(* CODESYS project sensata_lasermarker.library
   Company: Sensata Technologies
   DocFormat: reStructuredText
   Description: This library is for the Laser Markers.
   Version: 0.0.1
   Placeholder: Sensata_LaserMarker
   Title: Sensata_LaserMarker

Project tree, tasks and I/O mapping:
  libraries: Sensata_Common, * (Sensata Technologies); Sensata_Utilities, * (Sensata Technologies); Tc2_Standard, * (Beckhoff Automation GmbH); Tc2_System, * (Beckhoff Automation GmbH); Tc2_Utilities, * (Beckhoff Automation GmbH); Tc3_Module, * (Beckhoff Automation GmbH); Sensata_Vision, * (Sensata Technologies)
  Abstract/
    function block FB_LaserMarker [ST]
  Concrete/
    function block FB_KeyenceLaserMarkerMDX2000 [LD]: M_Connect, M_Disconnect, M_GetConnectStatus, P_bConnectBusy, P_bConnected, M_PeakCurrentProgram, M_GetCurrentProgram, M_GetProgramState, M_LoadProgram, M_PauseProgram, M_SaveCurrentLaserProgramtoPC, M_SendProgramtoLaser, M_StartMarking, M_StartProgram, M_StopMarking, M_StopProgram, M_UpdateProgramBlockInTheLaser, P_bProgramControlBusy, P_enumProgramState, P_strCurrentProgram, M_GetAllLaserErrorStatus, M_GetAllLaserStatus, M_ClearLaserErrors, M_Reset, P_bResetBusy, M_Trigger, P_bTriggerBusy, M_HandleCommand
  Interfaces/
    interface I_Markable: StartMarking, StopMarking
  Project Information/
    function F_GetCompany [ST]
    function F_GetTitle [ST]
    function F_GetVersion [ST]
  Version/
    global variables Global_Version
  global variables GVL_LaserMarker
*)

// Version/Global_Version
{attribute 'TcGenerated'}
{attribute 'no-analysis'}
{attribute 'linkalways'}
// This function has been automatically generated from the project information.
VAR_GLOBAL CONSTANT
	{attribute 'const_non_replaced'}
	stLibVersion_Sensata_LaserMarker : ST_LibVersion := (iMajor := 0, iMinor := 0, iBuild := 1, iRevision := 0, nFlags := 0, sVersion := '0.0.1');
END_VAR

// GVL_LaserMarker
VAR_GLOBAL
	LaserConnected : BOOL := FALSE;
	PeakCurrentProgramSuccess : BOOL := FALSE;
	SendProgramToLaserSuccess : BOOL := FALSE;
END_VAR

// Abstract/FB_LaserMarker
FUNCTION_BLOCK ABSTRACT FB_LaserMarker EXTENDS FB_Device
VAR_INPUT
END_VAR
VAR_OUTPUT
END_VAR
VAR
END_VAR

END_FUNCTION_BLOCK

// Concrete/FB_KeyenceLaserMarkerMDX2000
FUNCTION_BLOCK PUBLIC FB_KeyenceLaserMarkerMDX2000 EXTENDS FB_LaserMarker
	IMPLEMENTS 
		I_Connectable,
		I_Resettable,
		I_Programmable,
		I_Triggerable
VAR_INPUT
	fbApi : REFERENCE TO FB_AdsCommandRouter; (* Device API connection to the "". *)
END_VAR
VAR_OUTPUT
END_VAR
VAR
	// Connectable
	bApiConnected: BOOL; (* TRUE if the API is connected. *)
	bConnected: BOOL; (* TRUE if the Laser is connected. *)
	bConnecting: BOOL; (* TRUE while the connect command is running. *)
	bDisconnecting: BOOL; (* TRUE while the disconnect command is running. *)
	bActive: BOOL;
   bSendingSendLaserProgram : BOOL;
	
	//Laser Related Variables
	
	ADSRouter: Sensata_Utilities.FB_AdsCommandRouter;
END_VAR

// NETWORK 1

METHOD M_Connect : BOOL
VAR_INPUT
	
END_VAR
VAR_OUTPUT
	
END_VAR
VAR
	bApiResult: BOOL;
	arrParameters: T_ApiMethodParameters;
	bContinue: BOOL;
	bCommandResult: BOOL;
	bCommandSent: BOOL;
	strReturn: STRING(255);
	bMethodCalled: BOOL;
	udintErrorCode: UDINT;
	strErrorMessage: T_MaxString;
	strResult : T_MaxString;

    buildArray: BOOL;    
    doIt: BOOL;
    buildArrayDB: BOOL;
    tagName: STRING := 'strProc';
    sataType: STRING := 'String';
    arrParams: T_ApiParameterList;
    
    doReset: BOOL;
    
    strTarget: T_MaxString := 'Laser_1';//'PAC_1';
    strCommand: T_MaxString := 'Connect';//'Write';
//    strProc: T_MaxString := 'spInsert';
    
    paramDictionary : T_ApiParameterList;
    p1: T_MaxString := 'MyMachine';
    p2: T_MaxString := 'MyLocation';
    p3: T_MaxString := 'MyPC';



   strRet: T_MaxString;
    adsRouter: FB_AdsCommandRouter;
    bResult: BOOL;
    arrOutputs: T_ApiParameterList;
    bExecuted: BOOL;
    
    pBuilder: FB_ApiParamBuilder;
    pArray: Sensata_Utilities.UXINT;
//    stTest: ST_TestStruct;



END_VAR
//M_Connect := FALSE;
//IF NOT bApiConnected THEN
//	bApiConnected := fbApi.M_Connect();
//END_IF
//udintErrorCode := 100;
//strErrorMessage := 'Error While connecting to Laser Marker';

//IF bApiConnected THEN
//	IF NOT fbApi.P_bDeviceInterfaceBusy OR bActive THEN
//		// Set continue to true
//		bActive := TRUE;
		
//		// Send command to API
////		bApiResult := fbApi.M_CallMethod(THIS^.in_strUniqueId, 'ConnectToLaserMarker' , arrParameters, strReturn => strResult);
//		bApiResult := fbApi.M_CallMethod(THIS^.in_strUniqueId, 'Connect' , arrParameters, strReturn => strResult);
		
//		IF NOT fbApi.P_bDeviceInterfaceBusy THEN
//			// Set continue to false
//			bActive := FALSE;
			
//			// Throw an error if the API has an error
//			IF fbApi.P_bError THEN
//				THIS^.M_SetError(
//					udintErrorCode,
//					strErrorMessage);
//			// If result is successful, set results accordingly
//			ELSIF bApiResult AND GVL_LaserMarker.LaserConnected THEN
//				M_Connect := TRUE;
//			END_IF
//		END_IF
//	END_IF
//END_IF


//Copied from Sensata_Test (Aiswarya)
//IF NOT bApiConnected THEN
//	bApiConnected := fbApi.M_Connect();
//END_IF

//bCommandResult := THIS^.M_HandleCommand(
//	THIS^.in_strUniqueId,
//	'Connect',
//	arrParameters,
//	//E_VitrekV70_Error.Connect,
//	100,
//	'Error while trying to connect to laser!',
//	bConnecting,
//	bContinue => bContinue);

//M_Connect := FALSE;
//IF bContinue THEN
//	bConnecting := TRUE;
//ELSIF bCommandResult THEN
//	bConnected := TRUE;
//	M_Connect := TRUE;
//END_IF


//Kevin's new ADS Server logic


IF doReset THEN
    doReset := FALSE;
    doIt := FALSE;
    adsRouter.M_ClearError();
END_IF

IF buildArray THEN
    pBuilder.M_ClearParameters();
//    pBuilder.M_AddParameter('tName', tagName);
//    pBuilder.M_AddParameter('dType', sataType);
    //pBuilder.M_AddParameter('retObj', NULL);
    pBuilder.M_OutputToParameterList(arrParams);
    buildArray := FALSE;
END_IF

//IF buildArrayDB THEN
//    pBuilder.M_ClearParameters();
//    pBuilder.M_AddParameter('procName', strProc);
//    pArray := pBuilder.M_AddParameter('paramDictionary', stTest);
//    pBuilder.M_AddStructMember(pArray,'@MachineName',p1);
//    pBuilder.M_AddStructMember(pArray,'@Location',p2);
//    pBuilder.M_AddStructMember(pArray,'@PCName',p3);
//    pBuilder.M_OutputToParameterList(arrParams);
//    buildArrayDB := FALSE;
//END_IF

//strTarget is 'Laser_1' in this case
//strCommand is 'Connect' in this case
//arrParams needs to be built using array builder


IF doIt THEN
    bResult := adsRouter.M_RouteCommand
      (
        strTarget, 
        strCommand, 
        T#5S, 
        arrParams, 
        arrOutputs, 
        _out_bCommandExecuted => bExecuted, 
        _out_strReturnValue => strRet
      );
    IF bExecuted THEN
        doIt := FALSE;
    END_IF  
END_IF
END_METHOD

METHOD PUBLIC M_Disconnect : BOOL
VAR
	arrParameters : T_ApiMethodParameters;
	bCommandResult : BOOL;
	bContinue : BOOL;
	bApiResult: BOOL;
	udintErrorCode: UDINT;
	strReturn: STRING(255);
	strResult : T_MaxString;
	strErrorMessage: T_MaxString;
END_VAR
//M_Disconnect := FALSE;
//IF NOT bApiConnected THEN
//	bApiConnected := fbApi.M_Connect();
//END_IF

//udintErrorCode := 101;
//strErrorMessage := 'Error While Disconnecting from Laser Marker';

//IF bApiConnected THEN
//	IF NOT fbApi.P_bDeviceInterfaceBusy OR bActive THEN
//		// Set continue to true
//		bActive := TRUE;
		
//		// Send command to API
//		//bApiResult := fbApi.M_CallMethod(THIS^.in_strUniqueId, 'DisconnectFromLaserMarker' , arrParameters, strReturn => strResult);
//		bApiResult := fbApi.M_CallMethod(THIS^.in_strUniqueId, 'Disconnect' , arrParameters, strReturn => strResult);
		
//		IF NOT fbApi.P_bDeviceInterfaceBusy THEN
//			// Set continue to false
//			bActive := FALSE;
//			// Throw an error if the API has an error
//			IF fbApi.P_bError THEN
//				THIS^.M_SetError( udintErrorCode, strErrorMessage);
//			ELSIF bApiResult THEN // If result is successful, set results accordingly
//				M_Disconnect := TRUE;
//			END_IF
//		END_IF
//	END_IF
//END_IF
END_METHOD

{warning 'add method implementation '}
(* This method should explicitly check the connection status of the device.
	Once the connection status is known, this method should return TRUE.
	If this method fails, P_bConnected should be set to FALSE since the device
	is not absolutely known to still be connected. *)
METHOD M_GetConnectStatus : BOOL
VAR_OUTPUT
	(* This should return TRUE if all connections required to make the device
		function properly are known to be connected, and FALSE otherwise. *)
	bConnected	: BOOL;
END_VAR
bConnected := P_bConnected;
M_GetConnectStatus := TRUE;
THIS^.M_LogWarning('Get connect status not implemented in UR e-Series!');
END_METHOD

(* This property should be TRUE while any method in this interface is actively
	executing, or FALSE otherwise. *)
PROPERTY P_bConnectBusy : BOOL
GET
P_bConnectBusy := bConnecting OR bDisconnecting;
END_GET
END_PROPERTY

(* This should be set to TRUE if M_Connect is successful or M_GetConnectStatus
	determines the device to be connected, and set to FALSE if M_Disconnect is
	called at all, M_GetConnectStatus fails, or M_GetConnectStatus determines
	the device to be not connected. *)
PROPERTY P_bConnected : BOOL
GET
P_bConnected := bApiConnected AND bConnected;
END_GET
END_PROPERTY

METHOD PUBLIC M_PeakCurrentProgram : BOOL
VAR_INPUT
END_VAR
VAR
	arrParameters : T_ApiMethodParameters;
	bApiResult: BOOL;
	udintErrorCode: UDINT;
	strErrorMessage: T_MaxString;
	strResult: T_MaxString;
END_VAR
//M_PeakCurrentProgram := FALSE;
//IF NOT bApiConnected THEN
//	bApiConnected := fbApi.M_Connect();
//END_IF

//udintErrorCode := 300;
//strErrorMessage := 'Error While performing M_PeakCurrentProgram function with Laser Marker';

//IF bApiConnected THEN
//	IF NOT fbApi.P_bDeviceInterfaceBusy OR bActive THEN
//		// Set continue to true
//		bActive := TRUE;
//		// Send command to API
//		bApiResult := fbApi.M_CallMethod(THIS^.in_strUniqueId, 'PeakCurrentProgram' , arrParameters, strReturn => strResult);
		
//		IF NOT fbApi.P_bDeviceInterfaceBusy THEN
//			// Set continue to false
//			bActive := FALSE;
//			// Throw an error if the API has an error
//			IF fbApi.P_bError THEN
//				THIS^.M_SetError( udintErrorCode, strErrorMessage);
//			ELSIF bApiResult THEN // If result is successful, set results accordingly
//				M_PeakCurrentProgram := TRUE;
//			END_IF
//		END_IF
//	END_IF
//END_IF
END_METHOD

{warning 'add method implementation '}
(* This method should explicitly get the current program loaded on the device.
	If the current program is successfully gotten, this method should return
	TRUE and set P_strCurrentProgram and strCurrentProgram to the gotten
	program name. If this method fails, both should be set to empty strings. *)
METHOD M_GetCurrentProgram : BOOL
VAR_OUTPUT
	(* This should be set to the name of the currently loaded program if
		the method was successful, or a blank string otherwise. *)
	strCurrentProgram	: Sensata_Common.T_MaxString;
END_VAR
END_METHOD

{warning 'add method implementation '}
(* This method should explicitly check the program state of the device.
	Once the program state is known, this method should return TRUE and set
	P_enumProgramState and enumProgramState to the relevant E_ProgramState
	value, else it should set both to E_ProgramState.Unknown. *)
METHOD M_GetProgramState : BOOL
VAR_OUTPUT
	(* If the program state is successfully gotten, this should be set to
		the relevant E_ProgramState value. If this method fails, this should
		be set to E_ProgramState.Unknown. *)
	enumProgramState	: Sensata_Common.E_ProgramState;
END_VAR
END_METHOD

{warning 'add method implementation '}
(* This method should load a new program onto the device, and then return TRUE
	once program loading is completed. Once this method begins the program loading
	process, P_strCurrentProgram should be cleared unless it is still explicitly
	known to be loaded. *)
METHOD M_LoadProgram : BOOL
VAR_INPUT
	(* String representing the program to load. If string must be in a specific
		format, make sure to override this comment to document it. *)
	strProgram	: Sensata_Common.T_MaxString;
END_VAR
END_METHOD

{warning 'add method implementation '}
(* This program should move to the program state from whatever state it was in
	to the Paused state, and then return TRUE once successful. If the program
	state is Stopped, this method should return TRUE but keep the current state
	as Stopped, since Paused at the beginning at the program is equivalent to
	being Stopped. *)
METHOD M_PauseProgram : BOOL
END_METHOD

METHOD PUBLIC M_SaveCurrentLaserProgramtoPC : BOOL
VAR_INPUT
	LaserProgramFolderPath : STRING;
END_VAR
VAR
	arrParameters : T_ApiMethodParameters;
	bApiResult: BOOL;
	udintErrorCode: UDINT;
	strErrorMessage: T_MaxString;
	strResult: T_MaxString;
END_VAR
//M_SaveCurrentLaserProgramtoPC := FALSE;
//IF NOT bApiConnected THEN
//	bApiConnected := fbApi.M_Connect();
//END_IF

//udintErrorCode := 200;
//strErrorMessage := 'Error While performing M_SaveCurrentLaserProgramtoPC from Laser Marker';

//IF bApiConnected THEN
//	IF NOT fbApi.P_bDeviceInterfaceBusy OR bActive THEN
//		// Set continue to true
//		bActive := TRUE;
//		arrParameters[1][1] := 'LaserProgramFolderPath';
//		arrParameters[1][2] := LaserProgramFolderPath;
//		// Send command to API
//		bApiResult := fbApi.M_CallMethod(THIS^.in_strUniqueId, 'SendProgramtoLaser' , arrParameters, strReturn => strResult);
		
//		IF NOT fbApi.P_bDeviceInterfaceBusy THEN
//			// Set continue to false
//			bActive := FALSE;
//			// Throw an error if the API has an error
//			IF fbApi.P_bError THEN
//				THIS^.M_SetError( udintErrorCode, strErrorMessage);
//			ELSIF bApiResult THEN // If result is successful, set results accordingly
//				M_SaveCurrentLaserProgramtoPC := TRUE;
//			END_IF
//		END_IF
//	END_IF
//END_IF
END_METHOD

METHOD PUBLIC M_SendProgramtoLaser : BOOL
VAR_INPUT
	filepath : STRING;
	LaserMemoryLocation : INT;
END_VAR
VAR
	bApiResult: BOOL;
	arrParameters: T_ApiMethodParameters;
	strResult: T_MaxString;
	udintErrorCode: UDINT;
	strErrorMessage: T_MaxString;
	bCommandResult : BOOL;
    bContinue: BOOL;
END_VAR
////M_SendProgramtoLaser := FALSE;
////IF NOT bApiConnected THEN
////	bApiConnected := fbApi.M_Connect();
////END_IF

//udintErrorCode := 201;
//strErrorMessage := 'Error While performing M_SendProgramtoLaser from Laser Marker';

////IF bApiConnected THEN
////	IF NOT fbApi.P_bDeviceInterfaceBusy OR bActive THEN
////		// Set continue to true
////		bActive := TRUE;
////		arrParameters[1][1] := 'filepath';
////		arrParameters[1][2] := filepath;
////		arrParameters[2][1] := 'LaserMemoryLocation';
////		arrParameters[2][2] := TO_STRING(LaserMemoryLocation);
////		// Send command to API
////		bApiResult := fbApi.M_CallMethod(THIS^.in_strUniqueId, 'SendProgramtoLaser' , arrParameters, strReturn => strResult);
		
////		IF NOT fbApi.P_bDeviceInterfaceBusy THEN
////			// Set continue to false
////			bActive := FALSE;
////			// Throw an error if the API has an error
////			IF fbApi.P_bError THEN
////				THIS^.M_SetError( udintErrorCode, strErrorMessage);
////			ELSIF bApiResult AND GVL_LaserMarker.SendProgramToLaserSuccess THEN // If result is successful, set results accordingly
////				M_SendProgramtoLaser := TRUE;
////			END_IF
////		END_IF
////	END_IF
////END_IF


////Copied from Aish

//		arrParameters[1][1] := 'filepath';
//		arrParameters[1][2] := filepath;
//		arrParameters[2][1] := 'LaserMemoryLocation';
//		arrParameters[2][2] := TO_STRING(LaserMemoryLocation);

//bCommandResult := THIS^.M_HandleCommand(
//    THIS^.in_strUniqueId,
//    'SendProgramtoLaser',
//    arrParameters,
//    udintErrorCode,
//    strErrorMessage,
//    bSendingSendLaserProgram,
//    bContinue => bContinue);
//M_SendProgramtoLaser := FALSE;
//IF bContinue THEN
//    bSendingSendLaserProgram := TRUE;
//ELSIF bCommandResult THEN
//        M_SendProgramtoLaser := TRUE;
//END_IF
END_METHOD

METHOD PUBLIC M_StartMarking : BOOL
VAR_INPUT
END_VAR

VAR
	bApiResult: BOOL;
	arrParameters: T_ApiMethodParameters;
	strResult: T_MaxString;
	udintErrorCode: UDINT;
	strErrorMessage: T_MaxString;
END_VAR
//M_StartMarking := FALSE;
//IF NOT bApiConnected THEN
//	bApiConnected := fbApi.M_Connect();
//END_IF

//udintErrorCode := 202;
//strErrorMessage := 'Error While performing M_StartMarking from Laser Marker';

//IF bApiConnected THEN
//	IF NOT fbApi.P_bDeviceInterfaceBusy OR bActive THEN
//		// Set continue to true
//		bActive := TRUE;
//		// Send command to API
//		bApiResult := fbApi.M_CallMethod(THIS^.in_strUniqueId, 'StartMarking' , arrParameters, strReturn => strResult);
		
//		IF NOT fbApi.P_bDeviceInterfaceBusy THEN
//			// Set continue to false
//			bActive := FALSE;
//			// Throw an error if the API has an error
//			IF fbApi.P_bError THEN
//				THIS^.M_SetError( udintErrorCode, strErrorMessage);
//			ELSIF bApiResult THEN // If result is successful, set results accordingly
//				M_StartMarking := TRUE;
//			END_IF
//		END_IF
//	END_IF
//END_IF
END_METHOD

{warning 'add method implementation '}
(* This should move the program state from whatever state it is in to the
	Running state, and then return TRUE once successful. Starting from the
	Paused state should always continue execution from whatever point the
	program was at when the program was initially paused. *)
METHOD M_StartProgram : BOOL
END_METHOD

METHOD PUBLIC M_StopMarking : BOOL
VAR_INPUT
END_VAR
VAR
	bApiResult: BOOL;
	arrParameters: T_ApiMethodParameters;
	strResult: T_MaxString;
	udintErrorCode: UDINT;
	strErrorMessage: T_MaxString;
END_VAR
//M_StopMarking := FALSE;
//IF NOT bApiConnected THEN
//	bApiConnected := fbApi.M_Connect();
//END_IF

//udintErrorCode := 203;
//strErrorMessage := 'Error While performing M_StopMarking from Laser Marker';

//IF bApiConnected THEN
//	IF NOT fbApi.P_bDeviceInterfaceBusy OR bActive THEN
//		// Set continue to true
//		bActive := TRUE;
//		// Send command to API
//		bApiResult := fbApi.M_CallMethod(THIS^.in_strUniqueId, 'StopMarking' , arrParameters, strReturn => strResult);
		
//		IF NOT fbApi.P_bDeviceInterfaceBusy THEN
//			// Set continue to false
//			bActive := FALSE;
//			// Throw an error if the API has an error
//			IF fbApi.P_bError THEN
//				THIS^.M_SetError( udintErrorCode, strErrorMessage);
//			ELSIF bApiResult THEN // If result is successful, set results accordingly
//				M_StopMarking := TRUE;
//			END_IF
//		END_IF
//	END_IF
//END_IF
END_METHOD

{warning 'add method implementation '}
(* This should change the program state from whatever state it was in to the
	Stopped state and then return TRUE. Moving to the Stopped state should
	always reset the program execution back to the beginning. *)
METHOD M_StopProgram : BOOL
END_METHOD

METHOD PUBLIC M_UpdateProgramBlockInTheLaser : BOOL
VAR_INPUT
	LaserProgramMemoryLocation : INT;
	BlockNumber : INT;
	BlockData : STRING;
	BlockType : BlockTypes;
END_VAR
VAR
	bApiResult: BOOL;
	arrParameters: T_ApiMethodParameters;
	strResult: T_MaxString;
	udintErrorCode: UDINT;
	strErrorMessage: T_MaxString;
END_VAR
//M_UpdateProgramBlockInTheLaser := FALSE;
//IF NOT bApiConnected THEN
//	bApiConnected := fbApi.M_Connect();
//END_IF

//udintErrorCode := 204;
//strErrorMessage := 'Error While performing M_UpdateProgramBlockInTheLaser from Laser Marker';

//IF bApiConnected THEN
//	IF NOT fbApi.P_bDeviceInterfaceBusy OR bActive THEN
//		// Set continue to true
//		bActive := TRUE;
//		arrParameters[1][1] := 'LaserProgramMemoryLocation';
//		arrParameters[1][2] := TO_STRING(LaserProgramMemoryLocation);
//		arrParameters[2][1] := 'BlockNumber';
//		arrParameters[2][2] := TO_STRING(BlockNumber);
//		arrParameters[3][1] := 'BlockData';
//		arrParameters[3][2] := BlockData;
//		arrParameters[4][1] := 'BlockType';
//		arrParameters[4][2] := TO_STRING(BlockType);
		
//		// Send command to API
//		bApiResult := fbApi.M_CallMethod(THIS^.in_strUniqueId, 'UpdateSingleBlockInTheLaserProgram' , arrParameters, strReturn => strResult);
		
//		IF NOT fbApi.P_bDeviceInterfaceBusy THEN
//			// Set continue to false
//			bActive := FALSE;
//			// Throw an error if the API has an error
//			IF fbApi.P_bError THEN
//				THIS^.M_SetError( udintErrorCode, strErrorMessage);
//			ELSIF bApiResult THEN // If result is successful, set results accordingly
//				M_UpdateProgramBlockInTheLaser := TRUE;
//			END_IF
//		END_IF
//	END_IF
//END_IF
END_METHOD

(* This property should be TRUE while any method in this interface is actively
	executing, or FALSE otherwise. *)
PROPERTY P_bProgramControlBusy : BOOL
GET
END_GET
END_PROPERTY

(* The current E_ProgramState value of the device. This should be reset to
	E_ProgramState.Unknown if any methods in this interface interact with the
	device but fail. *)
PROPERTY P_enumProgramState : Sensata_Common.E_ProgramState
GET
END_GET
END_PROPERTY

(* The value of the currently loaded program. This should only be set by
	M_LoadProgram or M_GetCurrentProgram, and set to a blank string if either
	fail. *)
PROPERTY P_strCurrentProgram : Sensata_Common.T_MaxString
GET
END_GET
END_PROPERTY

METHOD PUBLIC M_GetAllLaserErrorStatus : BOOL
VAR_INPUT
END_VAR
END_METHOD

METHOD PUBLIC M_GetAllLaserStatus : BOOL
VAR_INPUT
END_VAR
END_METHOD

METHOD PUBLIC M_ClearLaserErrors : BOOL
VAR
	arrParameters : T_ApiMethodParameters;
	bApiResult: BOOL;
	udintErrorCode: UDINT;
//	strReturn: STRING(255);
	strResult : T_MaxString;
	strErrorMessage: T_MaxString;
END_VAR
//M_ClearLaserErrors := FALSE;
//IF NOT bApiConnected THEN
//	bApiConnected := fbApi.M_Connect();//What should we write here ? and should this be called for every function
//END_IF

//udintErrorCode := 400;
//strErrorMessage := 'Error While performing ClearLaserErrors on Laser Marker';

//IF bApiConnected THEN
//	IF NOT fbApi.P_bDeviceInterfaceBusy OR bActive THEN
//		// Set continue to true
//		bActive := TRUE;
		
//		// Send command to API
//		bApiResult := fbApi.M_CallMethod(THIS^.in_strUniqueId, 'ClearLaserErrors' , arrParameters, strReturn => strResult);
		
//		IF NOT fbApi.P_bDeviceInterfaceBusy THEN
//			// Set continue to false
//			bActive := FALSE;
//			// Throw an error if the API has an error
//			IF fbApi.P_bError THEN
//				THIS^.M_SetError( udintErrorCode, strErrorMessage);
//			ELSIF bApiResult THEN // If result is successful, set results accordingly
//				M_ClearLaserErrors := TRUE;
//			END_IF
//		END_IF
//	END_IF
//END_IF
END_METHOD

{warning 'add method implementation '}
(* This should clear any errors on the device and bring it to a state where
	it is ready to be energized or otherwise activated. *)
METHOD M_Reset : BOOL
END_METHOD

(* This property should be TRUE while any method in this interface is actively
	executing, or FALSE otherwise. *)
PROPERTY P_bResetBusy : BOOL
GET
END_GET
END_PROPERTY

{warning 'add method implementation '}
(*
Triggers the function block.
*)
METHOD M_Trigger : BOOL
END_METHOD

//{warning 'add property implementation'}
(*
Stays high while the function block is performing the tasks that were triggered.
*)
PROPERTY P_bTriggerBusy : BOOL
GET
END_GET
END_PROPERTY

METHOD PRIVATE M_HandleCommand : BOOL
VAR_INPUT
	strTarget:T_MaxString;
	strCommand: T_MaxString;
	arrParameters: T_ApiMethodParameters;
	udintErrorCode: UDINT;
	strErrorMessage: T_MaxString;
	bActive: BOOL;
END_VAR
VAR
	

END_VAR
VAR_OUTPUT
	bContinue: BOOL;
	strOutput: T_MaxString;
END_VAR

VAR
	bApiResult: BOOL;
END_VAR
//M_HandleCommand := FALSE;
//IF bApiConnected THEN
//	IF NOT fbApi.P_bDeviceInterfaceBusy OR bActive THEN
//		// Set continue to true
//		bContinue := TRUE;
		
//		// Send command to API
//		bApiResult := fbApi.M_CallMethod(strTarget,strCommand, arrParameters, strReturn => strOutput);
		
//		IF NOT fbApi.P_bDeviceInterfaceBusy THEN
//			// Set continue to false
//			bContinue := FALSE;
			
//			// Throw an error if the API has an error
//			IF fbApi.P_bError THEN
//				THIS^.M_SetError(
//					udintErrorCode,
//					strErrorMessage);
				
//			// If result is successful, set results accordingly
//			ELSIF bApiResult THEN
//				M_HandleCommand := TRUE;
//			END_IF
//		END_IF
//	END_IF
//END_IF
END_METHOD

END_FUNCTION_BLOCK

// Interfaces/I_Markable
INTERFACE I_Markable

METHOD StartMarking : BOOL
VAR_INPUT
END_VAR
END_METHOD

METHOD StopMarking : BOOL
VAR_INPUT
END_VAR
END_METHOD

END_INTERFACE

// Project Information/F_GetCompany
// This function has been automatically generated from the project information.
{attribute 'signature_flag' := '1073741824'}
{attribute 'TcGenerated'}
{attribute 'no-analysis'}
FUNCTION F_GetCompany : WSTRING
VAR_INPUT
	
END_VAR

F_GetCompany := "Sensata Technologies";

END_FUNCTION

// Project Information/F_GetTitle
// This function has been automatically generated from the project information.
{attribute 'signature_flag' := '1073741824'}
{attribute 'TcGenerated'}
{attribute 'no-analysis'}
FUNCTION F_GetTitle : WSTRING
VAR_INPUT
	
END_VAR

F_GetTitle := "Sensata_LaserMarker";

END_FUNCTION

// Project Information/F_GetVersion
// This function has been automatically generated from the project information.
{attribute 'signature_flag' := '1073741824'}
{attribute 'TcGenerated'}
{attribute 'no-analysis'}
FUNCTION F_GetVersion : ST_LibVersion
VAR_INPUT
	
END_VAR

F_GetVersion.iMajor := 0;
F_GetVersion.iMinor := 0;
F_GetVersion.iBuild := 1;
F_GetVersion.iRevision := 0;

END_FUNCTION
